{attribute 'qualified_only'}
{attribute 'strict'}
{attribute 'to_string'}
TYPE E_UnitStatus :
(
	Ok := 0,
	Error
);
END_TYPE

(* stored: Version 1.1.0.1
   DUT E_UnitStatus: Id {7300a613-bf84-4ecd-853a-38c28abb5007} *)
